DATA_BLOCK "DB2018_INST_M_SINA"
TITLE = DB2018_INST_M_SINA
{ S7_Optimized_Access := 'TRUE' }
AUTHOR : ABH
FAMILY : ZeusControl
VERSION : 1.0
NON_RETAIN
//Instancia bloque de funcion FB2017_M_SINA
"FB2017_ZC_M_SINA"

BEGIN
   Pulso1seg := FALSE;
   Simulacion := FALSE;
   Ack := FALSE;
   SeguridadesOK := TRUE;
   HWIDSTW[0] := 0;
   HWIDSTW[1] := 265;
   HWIDZSW[0] := 0;
   HWIDZSW[1] := 265;
   SinaSpeed[0].EnableAxis := FALSE;
   SinaSpeed[0].AckError := FALSE;
   SinaSpeed[0].SpeedSp := 0.0;
   SinaSpeed[0].RefSpeed := 0.0;
   SinaSpeed[0].ConfigAxis := 16#003F;
   SinaSpeed[0].HWIDSTW := 0;
   SinaSpeed[0].HWIDZSW := 0;
   SinaSpeed[0].AxisEnabled := FALSE;
   SinaSpeed[0].Lockout := FALSE;
   SinaSpeed[0].ActVelocity := 0.0;
   SinaSpeed[0].Error := FALSE;
   SinaSpeed[0].Status := 16#0000;
   SinaSpeed[0].DiagId := 16#0000;
   SinaSpeed[0].STW1 := 16#0000;
   SinaSpeed[0].VelocitySP := 16#0000;
   SinaSpeed[0].ZSW1 := 16#0000;
   SinaSpeed[0].VelocityAV := 16#0000;
   SinaSpeed[1].EnableAxis := FALSE;
   SinaSpeed[1].AckError := FALSE;
   SinaSpeed[1].SpeedSp := 0.0;
   SinaSpeed[1].RefSpeed := 100.0;
   SinaSpeed[1].ConfigAxis := 16#003F;
   SinaSpeed[1].HWIDSTW := 265;
   SinaSpeed[1].HWIDZSW := 265;
   SinaSpeed[1].AxisEnabled := FALSE;
   SinaSpeed[1].Lockout := FALSE;
   SinaSpeed[1].ActVelocity := 0.0;
   SinaSpeed[1].Error := FALSE;
   SinaSpeed[1].Status := 16#7002;
   SinaSpeed[1].DiagId := 16#0000;
   SinaSpeed[1].STW1 := 16#047E;
   SinaSpeed[1].VelocitySP := 16#0000;
   SinaSpeed[1].ZSW1 := 16#EB31;
   SinaSpeed[1].VelocityAV := 16#0000;

END_DATA_BLOCK

